% RSLogix 500 project Time How Long Something is ON.RSS, saved by version 10.00.00.00 %
PROJECT "UNTITLED"    % processor: Bul.1763 MicroLogix 1100 Series B %

PROGRAM FILES
  LAD 2   5 rungs

DATA FILES
  O0 OUTPUT  4 elements
  I1 INPUT  6 elements
  S2 STATUS  66 elements
  B3 BINARY  11 elements
  T4 TIMER  16 elements
  C5 COUNTER  1 elements
  R6 CONTROL  1 elements
  N7 INTEGER  1 elements
  F8 FLOAT  1 elements

LADDER 2
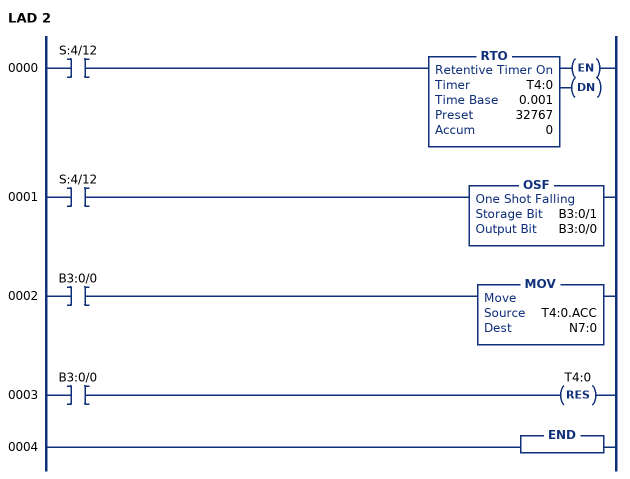
% Rung: 0 %
SOR XIC S:4/12 RTO T4:0 0.001 32767 0 EOR
% Rung: 1 %
SOR XIC S:4/12 OSF B3:0/1 B3:0/0 EOR
% Rung: 2 %
SOR XIC B3:0/0 MOV T4:0.ACC N7:0 EOR
% Rung: 3 %
SOR XIC B3:0/0 RES T4:0 EOR
% Rung: 4 %
SOR END EOR

DATA TABLE (non-zero values as saved)
DATA T4
% .PRE .ACC %
% T4:0 % 32767 0
% T4:15 % 10000 0
